TYPE stPoseGeneral :
STRUCT
	x : LREAL;
	y : LREAL;
	z: LREAL;
	rx: LREAL;
	ry: LREAL;
	rz: LREAL; //THETA
END_STRUCT
END_TYPE

(* stored: Version 1.1.0.1, ProductVersion 3.1.4026.18
   DUT stPoseGeneral: Id {e4f90f08-2c74-4a3a-b4af-3a5868a4d9f1} *)
